// Valid on Done (S3.12).
TYPE ST_SeparatorOutCmd :
STRUCT
    SeparateOk    : BOOL;
    SeparatorOpen : BOOL;
END_STRUCT
END_TYPE

(* stored: Version 1.1.0.1, ProductVersion 3.1.4024.12
   DUT ST_SeparatorOutCmd: Id {68fec8c6-2356-4470-88ec-eedcdc49f331} *)
